// TIA Portal V15 export
// export: Created 2019-02-04T15:20:19.8832449Z, ExportSetting WithDefaults, WithReadOnly, DisplayName Totally Integrated Automation Portal, DisplayVersion V15 Update 2, DisplayName TIA Portal Openness, DisplayVersion V15 Update 2, DisplayName STEP 7 Professional, DisplayVersion V15 Update 2, DisplayName STEP 7 Safety, DisplayVersion V15, DisplayName WinCC Professional, DisplayVersion V15 Update 2, DisplayName SIMATIC Visualization Architect, DisplayVersion V15 Update 1
FUNCTION "DESK_NAME_Call" : Void   // FC9, FBD
TITLE = DESK_NAME operating computer / DESK_NAME Bedienrechner
{ S7_Optimized_Access := 'FALSE' }
VERSION : 0.1
// stored: AutoNumber true, CodeModifiedDate 2019-02-04T15:19:08.6251442Z, CompileDate 2019-02-04T15:19:58.9716345Z, CreationDate 2016-08-15T15:32:48.1433866Z, HandleErrorsWithinBlock false, InterfaceModifiedDate 2016-02-03T14:10:29.6571349Z, IsConsistent true, IsIECCheckEnabled false, IsKnowHowProtected false, IsWriteProtected false, LibraryConformanceStatus Error: The block contains calls of single instances. Warning: The object contains access to global data blocks. Warning: The block contains direct access to inputs, outputs, bit memories, indirect access to the registry or indirect access to external memory areas that are unknown at the time of compilation., ModifiedDate 2019-02-04T15:19:08.6251442Z, ParameterModified 2016-02-03T14:10:29.6415099Z, PLCSimAdvancedSupport false, SetENOAutomatically False, StructureModified 2016-02-03T14:10:29.6571349Z, UDAEnableTagReadback false
BEGIN

REGION Network 1: Automatic start / Automatik Start
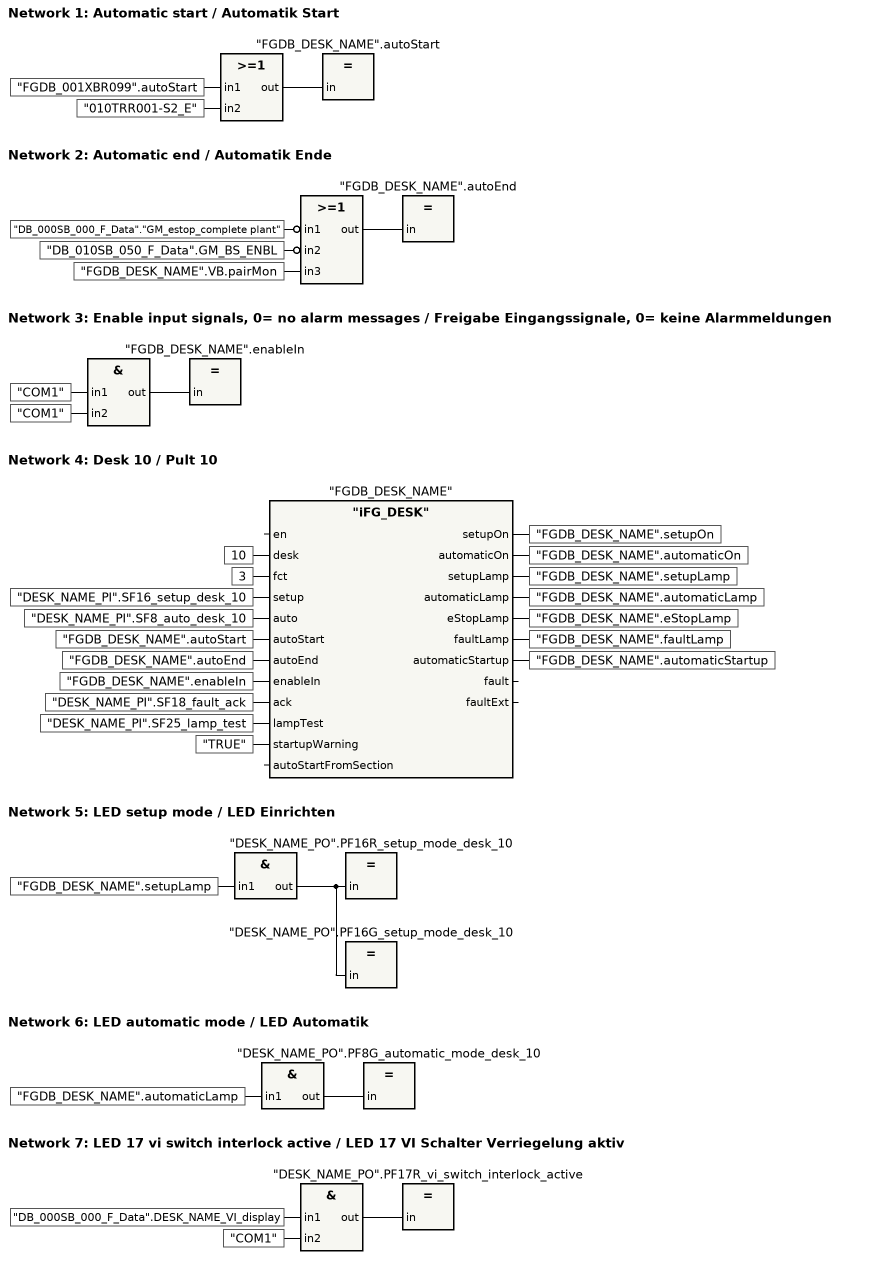
   "FGDB_DESK_NAME".autoStart := "FGDB_001XBR099".autoStart OR "010TRR001-S2_E";
END_REGION

REGION Network 2: Automatic end / Automatik Ende
   "FGDB_DESK_NAME".autoEnd := NOT "DB_000SB_000_F_Data"."GM_estop_complete plant" OR NOT "DB_010SB_050_F_Data".GM_BS_ENBL OR "FGDB_DESK_NAME".VB.pairMon;
END_REGION

REGION Network 3: Enable input signals, 0= no alarm messages / Freigabe Eingangssignale, 0= keine Alarmmeldungen
   "FGDB_DESK_NAME".enableIn := "COM1" AND "COM1";
END_REGION

REGION Network 4: Desk 10 / Pult 10
   "FGDB_DESK_NAME"(desk := 10,   // "iFG_DESK"
                    fct := 3,
                    setup := "DESK_NAME_PI".SF16_setup_desk_10,
                    auto := "DESK_NAME_PI".SF8_auto_desk_10,
                    autoStart := "FGDB_DESK_NAME".autoStart,
                    autoEnd := "FGDB_DESK_NAME".autoEnd,
                    enableIn := "FGDB_DESK_NAME".enableIn,
                    ack := "DESK_NAME_PI".SF18_fault_ack,
                    lampTest := "DESK_NAME_PI".SF25_lamp_test,
                    startupWarning := "TRUE",
                    setupOn => "FGDB_DESK_NAME".setupOn,
                    automaticOn => "FGDB_DESK_NAME".automaticOn,
                    setupLamp => "FGDB_DESK_NAME".setupLamp,
                    automaticLamp => "FGDB_DESK_NAME".automaticLamp,
                    eStopLamp => "FGDB_DESK_NAME".eStopLamp,
                    faultLamp => "FGDB_DESK_NAME".faultLamp,
                    automaticStartup => "FGDB_DESK_NAME".automaticStartup);
END_REGION

REGION Network 5: LED setup mode / LED Einrichten
   "DESK_NAME_PO".PF16R_setup_mode_desk_10 := "FGDB_DESK_NAME".setupLamp;
   "DESK_NAME_PO".PF16G_setup_mode_desk_10 := "FGDB_DESK_NAME".setupLamp;
END_REGION

REGION Network 6: LED automatic mode / LED Automatik
   "DESK_NAME_PO".PF8G_automatic_mode_desk_10 := "FGDB_DESK_NAME".automaticLamp;
END_REGION

REGION Network 7: LED 17 vi switch interlock active / LED 17 VI Schalter Verriegelung aktiv
   // COM1 -> Group message insert interlock local / COM1 -> Sammelmeldung Verriegelung Lokal einfügen
   "DESK_NAME_PO".PF17R_vi_switch_interlock_active := "DB_000SB_000_F_Data".DESK_NAME_VI_display AND "COM1";
END_REGION

REGION Network 8: LED fault / LED Störung
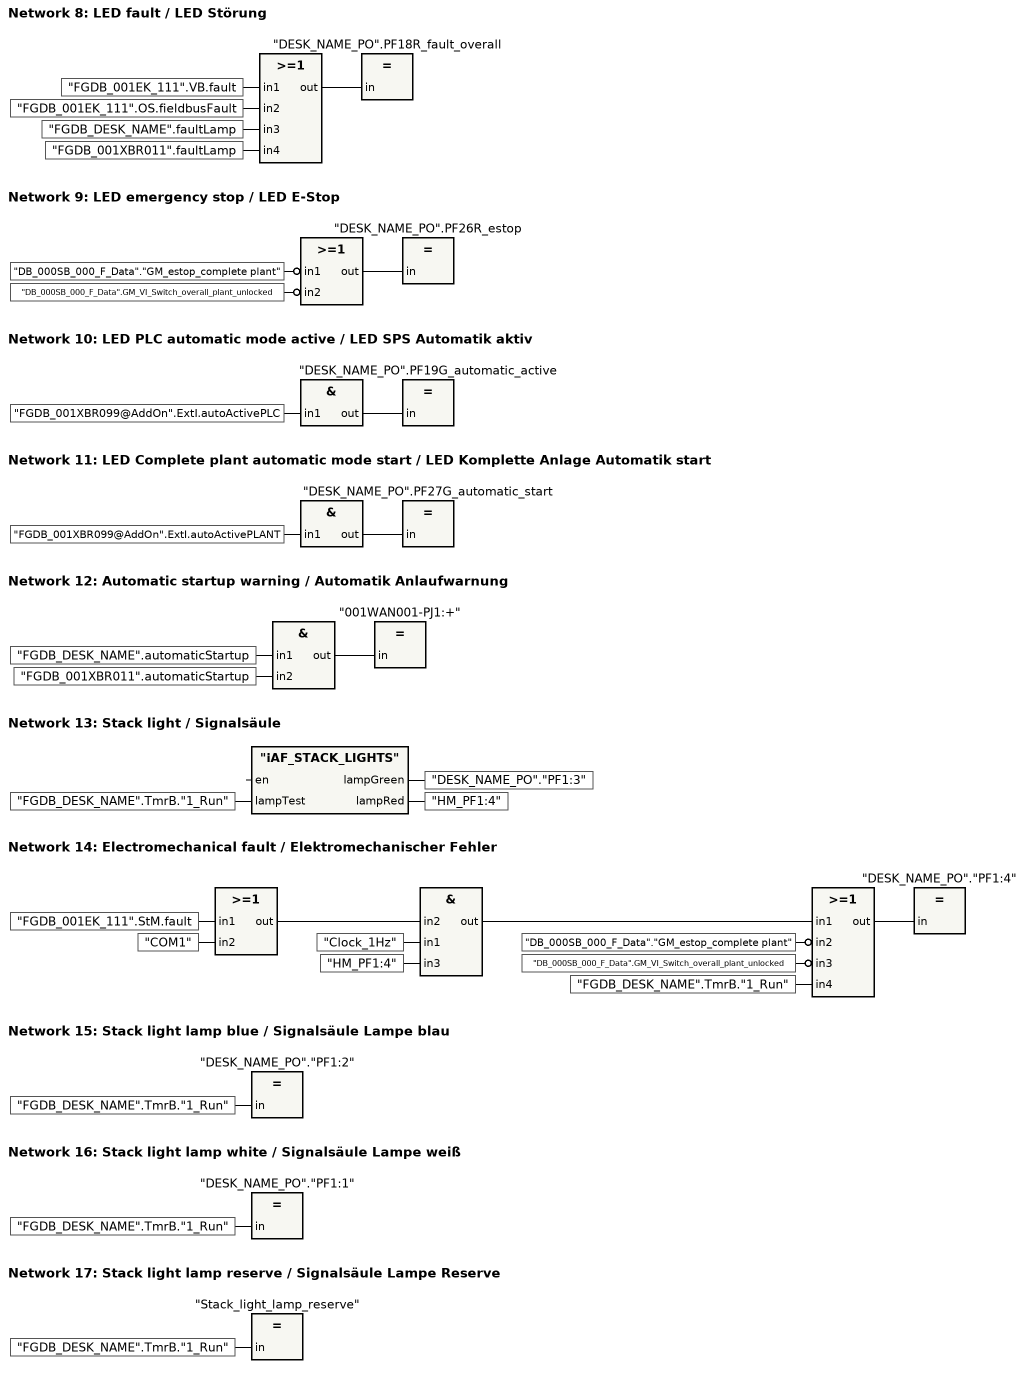
   "DESK_NAME_PO".PF18R_fault_overall := "FGDB_001EK_111".VB.fault OR "FGDB_001EK_111".OS.fieldbusFault OR "FGDB_DESK_NAME".faultLamp OR "FGDB_001XBR011".faultLamp;
END_REGION

REGION Network 9: LED emergency stop / LED E-Stop
   "DESK_NAME_PO".PF26R_estop := NOT "DB_000SB_000_F_Data"."GM_estop_complete plant" OR NOT "DB_000SB_000_F_Data".GM_VI_Switch_overall_plant_unlocked;
END_REGION

REGION Network 10: LED PLC automatic mode active / LED SPS Automatik aktiv
   "DESK_NAME_PO".PF19G_automatic_active := "FGDB_001XBR099@AddOn".ExtI.autoActivePLC;
END_REGION

REGION Network 11: LED Complete plant automatic mode start / LED Komplette Anlage Automatik start
   "DESK_NAME_PO".PF27G_automatic_start := "FGDB_001XBR099@AddOn".ExtI.autoActivePLANT;
END_REGION

REGION Network 12: Automatic startup warning / Automatik Anlaufwarnung
   "001WAN001-PJ1:+" := "FGDB_DESK_NAME".automaticStartup AND "FGDB_001XBR011".automaticStartup;
END_REGION

REGION Network 13: Stack light / Signalsäule
   "iAF_STACK_LIGHTS"(lampTest := "FGDB_DESK_NAME".TmrB."1_Run",
                      lampGreen => "DESK_NAME_PO"."PF1:3",
                      lampRed => "HM_PF1:4");
END_REGION

REGION Network 14: Electromechanical fault / Elektromechanischer Fehler
   "DESK_NAME_PO"."PF1:4" := (("FGDB_001EK_111".StM.fault OR "COM1") AND "Clock_1Hz" AND "HM_PF1:4") OR NOT "DB_000SB_000_F_Data"."GM_estop_complete plant" OR NOT "DB_000SB_000_F_Data".GM_VI_Switch_overall_plant_unlocked OR "FGDB_DESK_NAME".TmrB."1_Run";
END_REGION

REGION Network 15: Stack light lamp blue / Signalsäule Lampe blau
   "DESK_NAME_PO"."PF1:2" := "FGDB_DESK_NAME".TmrB."1_Run";
END_REGION

REGION Network 16: Stack light lamp white / Signalsäule Lampe weiß
   "DESK_NAME_PO"."PF1:1" := "FGDB_DESK_NAME".TmrB."1_Run";
END_REGION

REGION Network 17: Stack light lamp reserve / Signalsäule Lampe Reserve
   "Stack_light_lamp_reserve" := "FGDB_DESK_NAME".TmrB."1_Run";
END_REGION

REGION Network 18: Movement Screen / Bewegungsbild
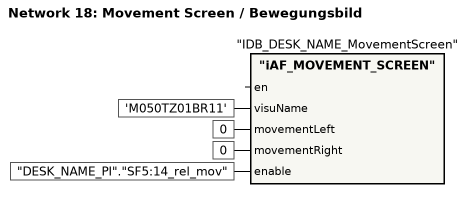
   "IDB_DESK_NAME_MovementScreen"(visuName := 'M050TZ01BR11',   // "iAF_MOVEMENT_SCREEN"
                           movementLeft := 0,
                           movementRight := 0,
                           enable := "DESK_NAME_PI"."SF5:14_rel_mov");
END_REGION
END_FUNCTION
